ABB RAPID module: Module1_plano.mod

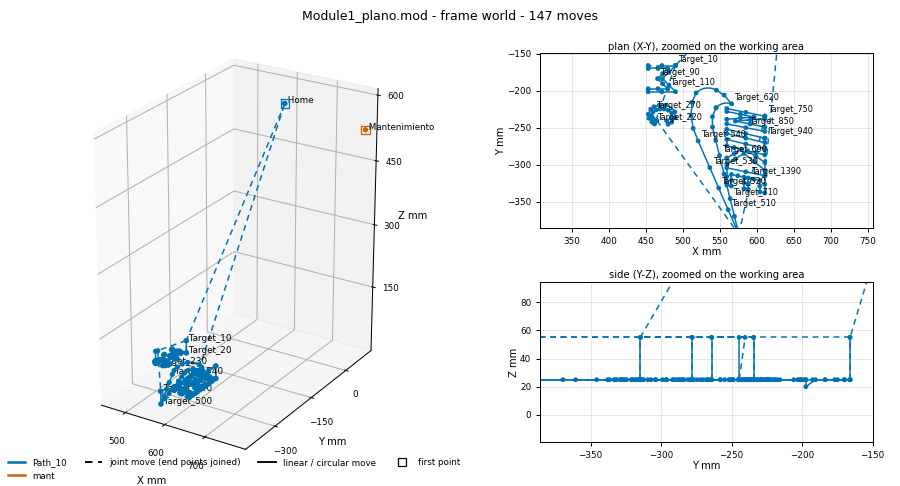
[picture p0: tool path of Module1_plano.mod in frame world, 147 of 147 moves have a stored position in this frame; points joined in program order, loops and branches not executed]
MODULE Module1
    PERS tooldata TCPTool_Lab1:=[TRUE,[[11.969,-5.577,162.232],[0.965925826,0,0.258819045,0]],[1,[0,0,1],[1,0,0,0],0,0,0]];
    TASK PERS wobjdata Workobject_2:=[FALSE,TRUE,"",[[667.5,-435,25],[0,0,1,0]],[[0,0,0],[1,0,0,0]]];
    CONST robtarget Target_10:=[[177.41,269.019,-30],[1,0,0,0],[0,0,-1,1],[9E+09,9E+09,9E+09,9E+09,9E+09,9E+09]];
    CONST robtarget Target_20:=[[177.41,269.019,0],[1,0,0,0],[0,0,-1,1],[9E+09,9E+09,9E+09,9E+09,9E+09,9E+09]];
    CONST robtarget Target_30:=[[195.844,269.019,0],[1,0,0,0],[0,0,-1,1],[9E+09,9E+09,9E+09,9E+09,9E+09,9E+09]];
    CONST robtarget Target_40:=[[214.279,269.019,0],[1,0,0,0],[0,0,-1,1],[9E+09,9E+09,9E+09,9E+09,9E+09,9E+09]];
    CONST robtarget Target_50:=[[214.279,265.019,0],[1,0,0,0],[0,0,-1,1],[9E+09,9E+09,9E+09,9E+09,9E+09,9E+09]];
    CONST robtarget Target_60:=[[201.112,265.019,0],[1,0,0,0],[0,0,-1,1],[9E+09,9E+09,9E+09,9E+09,9E+09,9E+09]];
    CONST robtarget Target_70:=[[187.944,265.019,0],[1,0,0,0],[0,0,-1,1],[9E+09,9E+09,9E+09,9E+09,9E+09,9E+09]];
    CONST robtarget Target_80:=[[194.783,258.18,0],[1,0,0,0],[0,0,-1,1],[9E+09,9E+09,9E+09,9E+09,9E+09,9E+09]];
    CONST robtarget Target_90:=[[201.622,251.341,0],[1,0,0,0],[0,0,-1,1],[9E+09,9E+09,9E+09,9E+09,9E+09,9E+09]];
    CONST robtarget Target_100:=[[194.783,244.503,0],[1,0,0,0],[0,0,-1,1],[9E+09,9E+09,9E+09,9E+09,9E+09,9E+09]];
    CONST robtarget Target_110:=[[187.944,237.664,5],[1,0,0,0],[0,0,-1,1],[9E+09,9E+09,9E+09,9E+09,9E+09,9E+09]];
    CONST robtarget Target_120:=[[201.112,237.664,0],[1,0,0,0],[0,0,-1,1],[9E+09,9E+09,9E+09,9E+09,9E+09,9E+09]];
    CONST robtarget Target_130:=[[214.279,237.664,0],[1,0,0,0],[0,0,-1,1],[9E+09,9E+09,9E+09,9E+09,9E+09,9E+09]];
    CONST robtarget Target_140:=[[214.279,233.664,0],[1,0,0,0],[0,0,-1,1],[9E+09,9E+09,9E+09,9E+09,9E+09,9E+09]];
    CONST robtarget Target_150:=[[195.844,233.664,0],[1,0,0,0],[0,0,-1,1],[9E+09,9E+09,9E+09,9E+09,9E+09,9E+09]];
    CONST robtarget Target_160:=[[177.41,233.664,0],[1,0,0,0],[0,0,-1,1],[9E+09,9E+09,9E+09,9E+09,9E+09,9E+09]];
    CONST robtarget Target_170:=[[186.248,242.503,0],[1,0,0,0],[0,0,-1,1],[9E+09,9E+09,9E+09,9E+09,9E+09,9E+09]];
    CONST robtarget Target_180:=[[195.087,251.341,0],[1,0,0,0],[0,0,-1,1],[9E+09,9E+09,9E+09,9E+09,9E+09,9E+09]];
    CONST robtarget Target_190:=[[186.248,260.18,0],[1,0,0,0],[0,0,-1,1],[9E+09,9E+09,9E+09,9E+09,9E+09,9E+09]];
    CONST robtarget Target_200:=[[177.41,269.019,0],[1,0,0,0],[0,0,-1,1],[9E+09,9E+09,9E+09,9E+09,9E+09,9E+09]];
    CONST robtarget Target_210:=[[177.41,269.019,-30],[1,0,0,0],[0,0,-1,1],[9E+09,9E+09,9E+09,9E+09,9E+09,9E+09]];
    CONST robtarget Target_220:=[[205.678,190.302,-30],[1,0,0,0],[0,0,-1,1],[9E+09,9E+09,9E+09,9E+09,9E+09,9E+09]];
    CONST robtarget Target_230:=[[205.623,190.276,0],[1,0,0,0],[0,0,-1,1],[9E+09,9E+09,9E+09,9E+09,9E+09,9E+09]];
    CONST robtarget Target_240:=[[202.955,194.702,0],[1,0,0,0],[0,0,-1,1],[9E+09,9E+09,9E+09,9E+09,9E+09,9E+09]];
    CONST robtarget Target_250:=[[207.34,197.113,0],[1,0,0,0],[0,0,-1,1],[9E+09,9E+09,9E+09,9E+09,9E+09,9E+09]];
    CONST robtarget Target_260:=[[209.847,201.03,0],[1,0,0,0],[0,0,-1,1],[9E+09,9E+09,9E+09,9E+09,9E+09,9E+09]];
    CONST robtarget Target_270:=[[208.011,206.295,0],[1,0,0,0],[0,0,-1,1],[9E+09,9E+09,9E+09,9E+09,9E+09,9E+09]];
    CONST robtarget Target_280:=[[203.511,209.124,0],[1,0,0,0],[0,0,-1,1],[9E+09,9E+09,9E+09,9E+09,9E+09,9E+09]];
    CONST robtarget Target_290:=[[198.638,210.318,0],[1,0,0,0],[0,0,-1,1],[9E+09,9E+09,9E+09,9E+09,9E+09,9E+09]];
    CONST robtarget Target_300:=[[192.941,210.304,0],[1,0,0,0],[0,0,-1,1],[9E+09,9E+09,9E+09,9E+09,9E+09,9E+09]];
    CONST robtarget Target_310:=[[187.344,208.773,0],[1,0,0,0],[0,0,-1,1],[9E+09,9E+09,9E+09,9E+09,9E+09,9E+09]];
    CONST robtarget Target_320:=[[182.65,205,0],[1,0,0,0],[0,0,-1,1],[9E+09,9E+09,9E+09,9E+09,9E+09,9E+09]];
    CONST robtarget Target_330:=[[182.874,198.696,0],[1,0,0,0],[0,0,-1,1],[9E+09,9E+09,9E+09,9E+09,9E+09,9E+09]];
    CONST robtarget Target_340:=[[189.379,194.489,0],[1,0,0,0],[0,0,-1,1],[9E+09,9E+09,9E+09,9E+09,9E+09,9E+09]];
    CONST robtarget Target_350:=[[187.41,189.702,0],[1,0,0,0],[0,0,-1,1],[9E+09,9E+09,9E+09,9E+09,9E+09,9E+09]];
    CONST robtarget Target_360:=[[182.414,192.529,0],[1,0,0,0],[0,0,-1,1],[9E+09,9E+09,9E+09,9E+09,9E+09,9E+09]];
    CONST robtarget Target_370:=[[178.043,198.417,0],[1,0,0,0],[0,0,-1,1],[9E+09,9E+09,9E+09,9E+09,9E+09,9E+09]];
    CONST robtarget Target_380:=[[178.344,206.368,0],[1,0,0,0],[0,0,-1,1],[9E+09,9E+09,9E+09,9E+09,9E+09,9E+09]];
    CONST robtarget Target_390:=[[182.556,211.614,0],[1,0,0,0],[0,0,-1,1],[9E+09,9E+09,9E+09,9E+09,9E+09,9E+09]];
    CONST robtarget Target_400:=[[190.831,215.342,0],[1,0,0,0],[0,0,-1,1],[9E+09,9E+09,9E+09,9E+09,9E+09,9E+09]];
    CONST robtarget Target_410:=[[199.222,215.629,0],[1,0,0,0],[0,0,-1,1],[9E+09,9E+09,9E+09,9E+09,9E+09,9E+09]];
    CONST robtarget Target_420:=[[206.382,213.378,0],[1,0,0,0],[0,0,-1,1],[9E+09,9E+09,9E+09,9E+09,9E+09,9E+09]];
    CONST robtarget Target_430:=[[210.902,210.005,0],[1,0,0,0],[0,0,-1,1],[9E+09,9E+09,9E+09,9E+09,9E+09,9E+09]];
    CONST robtarget Target_440:=[[214.199,203.307,0],[1,0,0,0],[0,0,-1,1],[9E+09,9E+09,9E+09,9E+09,9E+09,9E+09]];
    CONST robtarget Target_450:=[[213.42,197.838,0],[1,0,0,0],[0,0,-1,1],[9E+09,9E+09,9E+09,9E+09,9E+09,9E+09]];
    CONST robtarget Target_460:=[[209.362,192.6,0],[1,0,0,0],[0,0,-1,1],[9E+09,9E+09,9E+09,9E+09,9E+09,9E+09]];
    CONST robtarget Target_470:=[[205.915,190.416,0],[1,0,0,0],[0,0,-1,1],[9E+09,9E+09,9E+09,9E+09,9E+09,9E+09]];
    CONST robtarget Target_480:=[[202.627,194.59,-30],[1,0,0,0],[0,0,-1,1],[9E+09,9E+09,9E+09,9E+09,9E+09,9E+09]];
    CONST robtarget Target_490:=[[91.883,41.213,-30],[1,0,0,0],[-1,-1,0,1],[9E+09,9E+09,9E+09,9E+09,9E+09,9E+09]];
    CONST robtarget Target_500:=[[91.883,41.213,0],[1,0,0,0],[-1,-1,0,1],[9E+09,9E+09,9E+09,9E+09,9E+09,9E+09]];
    CONST robtarget Target_510:=[[106.332,74.333,0],[1,0,0,0],[-1,-1,0,1],[9E+09,9E+09,9E+09,9E+09,9E+09,9E+09]];
    CONST robtarget Target_520:=[[119.103,103.607,0],[1,0,0,0],[-1,-1,0,1],[9E+09,9E+09,9E+09,9E+09,9E+09,9E+09]];
    CONST robtarget Target_530:=[[131.177,131.283,0],[1,0,0,0],[0,0,-1,1],[9E+09,9E+09,9E+09,9E+09,9E+09,9E+09]];
    CONST robtarget Target_540:=[[146.843,167.193,0],[1,0,0,0],[0,0,-1,1],[9E+09,9E+09,9E+09,9E+09,9E+09,9E+09]];
    CONST robtarget Target_550:=[[153.569,184.183,0],[1,0,0,0],[0,0,-1,1],[9E+09,9E+09,9E+09,9E+09,9E+09,9E+09]];
    CONST robtarget Target_560:=[[156.337,201.217,0],[1,0,0,0],[0,0,-1,1],[9E+09,9E+09,9E+09,9E+09,9E+09,9E+09]];
    CONST robtarget Target_570:=[[155.288,219.26,0],[1,0,0,0],[0,0,-1,1],[9E+09,9E+09,9E+09,9E+09,9E+09,9E+09]];
    CONST robtarget Target_580:=[[149.597,231.965,0],[1,0,0,0],[0,0,-1,1],[9E+09,9E+09,9E+09,9E+09,9E+09,9E+09]];
    CONST robtarget Target_590:=[[140.915,237.42,0],[1,0,0,0],[0,0,-1,1],[9E+09,9E+09,9E+09,9E+09,9E+09,9E+09]];
    CONST robtarget Target_600:=[[122.252,235.701,0],[1,0,0,0],[0,0,-1,1],[9E+09,9E+09,9E+09,9E+09,9E+09,9E+09]];
    CONST robtarget Target_610:=[[111.771,229.081,0],[1,0,0,0],[0,0,-1,1],[9E+09,9E+09,9E+09,9E+09,9E+09,9E+09]];
    CONST robtarget Target_620:=[[101.618,217.264,0],[1,0,0,0],[0,0,-1,1],[9E+09,9E+09,9E+09,9E+09,9E+09,9E+09]];
    CONST robtarget Target_630:=[[112.39,217.915,0],[1,0,0,0],[0,0,-1,1],[9E+09,9E+09,9E+09,9E+09,9E+09,9E+09]];
    CONST robtarget Target_640:=[[122.65,212.032,0],[1,0,0,0],[0,0,-1,1],[9E+09,9E+09,9E+09,9E+09,9E+09,9E+09]];
    CONST robtarget Target_650:=[[122.562,212.129,0],[1,0,0,0],[0,0,-1,1],[9E+09,9E+09,9E+09,9E+09,9E+09,9E+09]];
    CONST robtarget Target_660:=[[127.578,199.979,0],[1,0,0,0],[0,0,-1,1],[9E+09,9E+09,9E+09,9E+09,9E+09,9E+09]];
    CONST robtarget Target_670:=[[127.52,186.008,0],[1,0,0,0],[0,0,-1,1],[9E+09,9E+09,9E+09,9E+09,9E+09,9E+09]];
    CONST robtarget Target_680:=[[123.036,167.787,0],[1,0,0,0],[0,0,-1,1],[9E+09,9E+09,9E+09,9E+09,9E+09,9E+09]];
    CONST robtarget Target_690:=[[118.036,147.473,0],[1,0,0,0],[0,0,-1,1],[9E+09,9E+09,9E+09,9E+09,9E+09,9E+09]];
    CONST robtarget Target_700:=[[111.892,122.51,0],[1,0,0,0],[-1,-1,0,1],[9E+09,9E+09,9E+09,9E+09,9E+09,9E+09]];
    CONST robtarget Target_710:=[[103.706,89.25,0],[1,0,0,0],[-1,-1,0,1],[9E+09,9E+09,9E+09,9E+09,9E+09,9E+09]];
    CONST robtarget Target_720:=[[97.833,65.387,0],[1,0,0,0],[-1,-1,0,1],[9E+09,9E+09,9E+09,9E+09,9E+09,9E+09]];
    CONST robtarget Target_730:=[[91.883,41.213,0],[1,0,0,0],[-1,-1,0,1],[9E+09,9E+09,9E+09,9E+09,9E+09,9E+09]];
    CONST robtarget Target_740:=[[91.883,41.213,-30],[1,0,0,0],[-1,-1,0,1],[9E+09,9E+09,9E+09,9E+09,9E+09,9E+09]];
    CONST robtarget Target_750:=[[56.869,200.624,-30],[1,0,0,0],[0,0,-1,1],[9E+09,9E+09,9E+09,9E+09,9E+09,9E+09]];
    CONST robtarget Target_760:=[[56.869,200.624,0],[1,0,0,0],[0,0,-1,1],[9E+09,9E+09,9E+09,9E+09,9E+09,9E+09]];
    CONST robtarget Target_770:=[[82.551,205.76,0],[1,0,0,0],[0,0,-1,1],[9E+09,9E+09,9E+09,9E+09,9E+09,9E+09]];
    CONST robtarget Target_780:=[[108.233,210.896,0],[1,0,0,0],[0,0,-1,1],[9E+09,9E+09,9E+09,9E+09,9E+09,9E+09]];
    CONST robtarget Target_790:=[[108.233,206.964,0],[1,0,0,0],[0,0,-1,1],[9E+09,9E+09,9E+09,9E+09,9E+09,9E+09]];
    CONST robtarget Target_800:=[[89.785,203.274,0],[1,0,0,0],[0,0,-1,1],[9E+09,9E+09,9E+09,9E+09,9E+09,9E+09]];
    CONST robtarget Target_810:=[[71.337,199.585,0],[1,0,0,0],[0,0,-1,1],[9E+09,9E+09,9E+09,9E+09,9E+09,9E+09]];
    CONST robtarget Target_820:=[[89.785,198.008,0],[1,0,0,0],[0,0,-1,1],[9E+09,9E+09,9E+09,9E+09,9E+09,9E+09]];
    CONST robtarget Target_830:=[[108.233,196.431,0],[1,0,0,0],[0,0,-1,1],[9E+09,9E+09,9E+09,9E+09,9E+09,9E+09]];
    CONST robtarget Target_840:=[[108.233,190.27,0],[1,0,0,0],[0,0,-1,1],[9E+09,9E+09,9E+09,9E+09,9E+09,9E+09]];
    CONST robtarget Target_850:=[[82.554,185.135,0],[1,0,0,0],[0,0,-1,1],[9E+09,9E+09,9E+09,9E+09,9E+09,9E+09]];
    CONST robtarget Target_860:=[[56.875,179.999,0],[1,0,0,0],[0,0,-1,1],[9E+09,9E+09,9E+09,9E+09,9E+09,9E+09]];
    CONST robtarget Target_870:=[[56.875,186.086,0],[1,0,0,0],[0,0,-1,1],[9E+09,9E+09,9E+09,9E+09,9E+09,9E+09]];
    CONST robtarget Target_880:=[[76.742,190.059,0],[1,0,0,0],[0,0,-1,1],[9E+09,9E+09,9E+09,9E+09,9E+09,9E+09]];
    CONST robtarget Target_890:=[[96.61,194.033,0],[1,0,0,0],[0,0,-1,1],[9E+09,9E+09,9E+09,9E+09,9E+09,9E+09]];
    CONST robtarget Target_900:=[[76.742,195.731,0],[1,0,0,0],[0,0,-1,1],[9E+09,9E+09,9E+09,9E+09,9E+09,9E+09]];
    CONST robtarget Target_910:=[[56.875,197.429,0],[1,0,0,0],[0,0,-1,1],[9E+09,9E+09,9E+09,9E+09,9E+09,9E+09]];
    CONST robtarget Target_920:=[[56.869,200.624,0],[1,0,0,0],[0,0,-1,1],[9E+09,9E+09,9E+09,9E+09,9E+09,9E+09]];
    CONST robtarget Target_930:=[[56.869,200.624,-30],[1,0,0,0],[0,0,-1,1],[9E+09,9E+09,9E+09,9E+09,9E+09,9E+09]];
    CONST robtarget Target_940:=[[56.875,170.875,-30],[1,0,0,0],[0,0,-1,1],[9E+09,9E+09,9E+09,9E+09,9E+09,9E+09]];
    CONST robtarget Target_950:=[[56.875,170.875,0],[1,0,0,0],[0,0,-1,1],[9E+09,9E+09,9E+09,9E+09,9E+09,9E+09]];
    CONST robtarget Target_960:=[[82.554,176.959,0],[1,0,0,0],[0,0,-1,1],[9E+09,9E+09,9E+09,9E+09,9E+09,9E+09]];
    CONST robtarget Target_970:=[[108.233,183.043,0],[1,0,0,0],[0,0,-1,1],[9E+09,9E+09,9E+09,9E+09,9E+09,9E+09]];
    CONST robtarget Target_980:=[[108.233,177.043,0],[1,0,0,0],[0,0,-1,1],[9E+09,9E+09,9E+09,9E+09,9E+09,9E+09]];
    CONST robtarget Target_990:=[[82.554,170.959,0],[1,0,0,0],[0,0,-1,1],[9E+09,9E+09,9E+09,9E+09,9E+09,9E+09]];
    CONST robtarget Target_1000:=[[56.875,164.875,0],[1,0,0,0],[0,0,-1,1],[9E+09,9E+09,9E+09,9E+09,9E+09,9E+09]];
    CONST robtarget Target_1010:=[[56.875,170.875,0],[1,0,0,0],[0,0,-1,1],[9E+09,9E+09,9E+09,9E+09,9E+09,9E+09]];
    CONST robtarget Target_1020:=[[56.875,170.875,-30],[1,0,0,0],[0,0,-1,1],[9E+09,9E+09,9E+09,9E+09,9E+09,9E+09]];
    CONST robtarget Target_1030:=[[56.875,157.002,-30],[1,0,0,0],[0,0,-1,1],[9E+09,9E+09,9E+09,9E+09,9E+09,9E+09]];
    CONST robtarget Target_1040:=[[56.875,157.002,0],[1,0,0,0],[0,0,-1,1],[9E+09,9E+09,9E+09,9E+09,9E+09,9E+09]];
    CONST robtarget Target_1050:=[[82.554,163.085,0],[1,0,0,0],[0,0,-1,1],[9E+09,9E+09,9E+09,9E+09,9E+09,9E+09]];
    CONST robtarget Target_1060:=[[108.233,169.169,0],[1,0,0,0],[0,0,-1,1],[9E+09,9E+09,9E+09,9E+09,9E+09,9E+09]];
    CONST robtarget Target_1070:=[[108.233,160.652,0],[1,0,0,0],[0,0,-1,1],[9E+09,9E+09,9E+09,9E+09,9E+09,9E+09]];
    CONST robtarget Target_1080:=[[98.214,158.278,0],[1,0,0,0],[0,0,-1,1],[9E+09,9E+09,9E+09,9E+09,9E+09,9E+09]];
    CONST robtarget Target_1090:=[[88.195,155.905,0],[1,0,0,0],[0,0,-1,1],[9E+09,9E+09,9E+09,9E+09,9E+09,9E+09]];
    CONST robtarget Target_1100:=[[98.214,150.082,0],[1,0,0,0],[0,0,-1,1],[9E+09,9E+09,9E+09,9E+09,9E+09,9E+09]];
    CONST robtarget Target_1110:=[[108.233,144.259,0],[1,0,0,0],[0,0,-1,1],[9E+09,9E+09,9E+09,9E+09,9E+09,9E+09]];
    CONST robtarget Target_1120:=[[108.233,135.914,0],[1,0,0,0],[0,0,-1,1],[9E+09,9E+09,9E+09,9E+09,9E+09,9E+09]];
    CONST robtarget Target_1130:=[[96.587,143.111,0],[1,0,0,0],[0,0,-1,1],[9E+09,9E+09,9E+09,9E+09,9E+09,9E+09]];
    CONST robtarget Target_1140:=[[84.942,150.308,0],[1,0,0,0],[0,0,-1,1],[9E+09,9E+09,9E+09,9E+09,9E+09,9E+09]];
    CONST robtarget Target_1150:=[[70.909,139.04,0],[1,0,0,0],[0,0,-1,1],[9E+09,9E+09,9E+09,9E+09,9E+09,9E+09]];
    CONST robtarget Target_1160:=[[56.875,127.772,0],[1,0,0,0],[-1,-1,0,1],[9E+09,9E+09,9E+09,9E+09,9E+09,9E+09]];
    CONST robtarget Target_1170:=[[56.875,138.348,0],[1,0,0,0],[0,0,-1,1],[9E+09,9E+09,9E+09,9E+09,9E+09,9E+09]];
    CONST robtarget Target_1180:=[[68.658,146.208,0],[1,0,0,0],[0,0,-1,1],[9E+09,9E+09,9E+09,9E+09,9E+09,9E+09]];
    CONST robtarget Target_1190:=[[80.44,154.068,0],[1,0,0,0],[0,0,-1,1],[9E+09,9E+09,9E+09,9E+09,9E+09,9E+09]];
    CONST robtarget Target_1200:=[[68.658,151.276,0],[1,0,0,0],[0,0,-1,1],[9E+09,9E+09,9E+09,9E+09,9E+09,9E+09]];
    CONST robtarget Target_1210:=[[56.875,148.485,0],[1,0,0,0],[0,0,-1,1],[9E+09,9E+09,9E+09,9E+09,9E+09,9E+09]];
    CONST robtarget Target_1220:=[[56.875,157.002,0],[1,0,0,0],[0,0,-1,1],[9E+09,9E+09,9E+09,9E+09,9E+09,9E+09]];
    CONST robtarget Target_1230:=[[56.875,157.002,-30],[1,0,0,0],[0,0,-1,1],[9E+09,9E+09,9E+09,9E+09,9E+09,9E+09]];
    CONST robtarget Target_1240:=[[56.875,120.255,-30],[1,0,0,0],[-1,-1,0,1],[9E+09,9E+09,9E+09,9E+09,9E+09,9E+09]];
    CONST robtarget Target_1250:=[[56.875,120.255,0],[1,0,0,0],[-1,-1,0,1],[9E+09,9E+09,9E+09,9E+09,9E+09,9E+09]];
    CONST robtarget Target_1260:=[[82.554,125.558,0],[1,0,0,0],[-1,-1,0,1],[9E+09,9E+09,9E+09,9E+09,9E+09,9E+09]];
    CONST robtarget Target_1270:=[[108.233,130.861,0],[1,0,0,0],[0,0,-1,1],[9E+09,9E+09,9E+09,9E+09,9E+09,9E+09]];
    CONST robtarget Target_1280:=[[108.233,119.251,0],[1,0,0,0],[-1,-1,0,1],[9E+09,9E+09,9E+09,9E+09,9E+09,9E+09]];
    CONST robtarget Target_1290:=[[108.233,107.642,0],[1,0,0,0],[-1,-1,0,1],[9E+09,9E+09,9E+09,9E+09,9E+09,9E+09]];
    CONST robtarget Target_1300:=[[101.866,106.328,0],[1,0,0,0],[-1,-1,0,1],[9E+09,9E+09,9E+09,9E+09,9E+09,9E+09]];
    CONST robtarget Target_1310:=[[101.866,114.138,0],[1,0,0,0],[-1,-1,0,1],[9E+09,9E+09,9E+09,9E+09,9E+09,9E+09]];
    CONST robtarget Target_1320:=[[101.866,121.949,0],[1,0,0,0],[-1,-1,0,1],[9E+09,9E+09,9E+09,9E+09,9E+09,9E+09]];
    CONST robtarget Target_1330:=[[93.404,120.169,0],[1,0,0,0],[-1,-1,0,1],[9E+09,9E+09,9E+09,9E+09,9E+09,9E+09]];
    CONST robtarget Target_1340:=[[84.942,118.39,0],[1,0,0,0],[-1,-1,0,1],[9E+09,9E+09,9E+09,9E+09,9E+09,9E+09]];
    CONST robtarget Target_1350:=[[84.942,110.611,0],[1,0,0,0],[-1,-1,0,1],[9E+09,9E+09,9E+09,9E+09,9E+09,9E+09]];
    CONST robtarget Target_1360:=[[84.942,102.833,0],[1,0,0,0],[-1,-1,0,1],[9E+09,9E+09,9E+09,9E+09,9E+09,9E+09]];
    CONST robtarget Target_1370:=[[79.224,101.652,0],[1,0,0,0],[-1,-1,0,1],[9E+09,9E+09,9E+09,9E+09,9E+09,9E+09]];
    CONST robtarget Target_1380:=[[79.224,109.42,0],[1,0,0,0],[-1,-1,0,1],[9E+09,9E+09,9E+09,9E+09,9E+09,9E+09]];
    CONST robtarget Target_1390:=[[79.224,117.187,0],[1,0,0,0],[-1,-1,0,1],[9E+09,9E+09,9E+09,9E+09,9E+09,9E+09]];
    CONST robtarget Target_1400:=[[71.411,115.544,0],[1,0,0,0],[-1,-1,0,1],[9E+09,9E+09,9E+09,9E+09,9E+09,9E+09]];
    CONST robtarget Target_1410:=[[63.597,113.901,0],[1,0,0,0],[-1,-1,0,1],[9E+09,9E+09,9E+09,9E+09,9E+09,9E+09]];
    CONST robtarget Target_1420:=[[63.597,106.163,0],[1,0,0,0],[-1,-1,0,1],[9E+09,9E+09,9E+09,9E+09,9E+09,9E+09]];
    CONST robtarget Target_1430:=[[63.597,98.425,0],[1,0,0,0],[-1,-1,0,1],[9E+09,9E+09,9E+09,9E+09,9E+09,9E+09]];
    CONST robtarget Target_1440:=[[56.875,97.037,0],[1,0,0,0],[-1,-1,0,1],[9E+09,9E+09,9E+09,9E+09,9E+09,9E+09]];
    CONST robtarget Target_1450:=[[56.875,108.646,0],[1,0,0,0],[-1,-1,0,1],[9E+09,9E+09,9E+09,9E+09,9E+09,9E+09]];
    CONST robtarget Target_1460:=[[56.875,120.255,0],[1,0,0,0],[-1,-1,0,1],[9E+09,9E+09,9E+09,9E+09,9E+09,9E+09]];
    CONST robtarget Target_1470:=[[56.875,120.255,-30],[1,0,0,0],[-1,-1,0,1],[9E+09,9E+09,9E+09,9E+09,9E+09,9E+09]];
    CONST robtarget Home:=[[26.695815447,429.423,-563.018541942],[0.965925826,0,-0.258819045,0],[-1,0,-1,0],[9E+09,9E+09,9E+09,9E+09,9E+09,9E+09]];
    CONST robtarget Home_2:=[[74.783200826,129.426583542,-420.91739945],[0.993217397,0.000004228,0.116272108,0.000000495],[0,1,-2,1],[9E+09,9E+09,9E+09,9E+09,9E+09,9E+09]];
    CONST robtarget Mantenimiento:=[[-116.188,526.934,-500.556],[0.924164952,-0.278371196,-0.154994418,-0.210725769],[0,0,-1,0],[9E+09,9E+09,9E+09,9E+09,9E+09,9E+09]];
    CONST robtarget Home_1:=[[-77.086561778,129.419166281,-428.818733092],[0.993216571,-0.00000444,0.11627916,-0.00000052],[-1,0,-1,0],[9E+09,9E+09,9E+09,9E+09,9E+09,9E+09]];

    PROC Path_10()
        MoveJ Home,v200,z5,TCPTool_Lab1\WObj:=Workobject_2;
        MoveJ Target_10,v200,z5,TCPTool_Lab1\WObj:=Workobject_2;
        MoveL Target_20,v200,fine,TCPTool_Lab1\WObj:=Workobject_2;
        MoveL Target_30,v100,z0,TCPTool_Lab1\WObj:=Workobject_2;
        MoveJ Target_40,v100,z0,TCPTool_Lab1\WObj:=Workobject_2;
        MoveL Target_50,v100,z0,TCPTool_Lab1\WObj:=Workobject_2;
        MoveL Target_60,v100,z0,TCPTool_Lab1\WObj:=Workobject_2;
        MoveL Target_70,v100,z0,TCPTool_Lab1\WObj:=Workobject_2;
        MoveL Target_80,v100,z0,TCPTool_Lab1\WObj:=Workobject_2;
        MoveL Target_90,v100,z0,TCPTool_Lab1\WObj:=Workobject_2;
        MoveL Target_100,v100,z0,TCPTool_Lab1\WObj:=Workobject_2;
        MoveL Target_110,v100,z0,TCPTool_Lab1\WObj:=Workobject_2;
        MoveL Target_120,v100,z0,TCPTool_Lab1\WObj:=Workobject_2;
        MoveL Target_130,v100,z0,TCPTool_Lab1\WObj:=Workobject_2;
        MoveL Target_140,v100,z0,TCPTool_Lab1\WObj:=Workobject_2;
        MoveL Target_150,v100,z0,TCPTool_Lab1\WObj:=Workobject_2;
        MoveL Target_160,v100,z0,TCPTool_Lab1\WObj:=Workobject_2;
        MoveL Target_170,v100,z0,TCPTool_Lab1\WObj:=Workobject_2;
        MoveL Target_180,v100,z0,TCPTool_Lab1\WObj:=Workobject_2;
        MoveL Target_190,v100,z0,TCPTool_Lab1\WObj:=Workobject_2;
        MoveL Target_200,v100,z0,TCPTool_Lab1\WObj:=Workobject_2;
        MoveJ Target_210,v200,z5,TCPTool_Lab1\WObj:=Workobject_2;
        MoveJ Target_220,v200,z5,TCPTool_Lab1\WObj:=Workobject_2;
        MoveL Target_230,v100,fine,TCPTool_Lab1\WObj:=Workobject_2;
        MoveL Target_240,v100,z0,TCPTool_Lab1\WObj:=Workobject_2;
        MoveL Target_250,v100,z0,TCPTool_Lab1\WObj:=Workobject_2;
        MoveL Target_260,v100,z0,TCPTool_Lab1\WObj:=Workobject_2;
        MoveL Target_270,v100,z0,TCPTool_Lab1\WObj:=Workobject_2;
        MoveL Target_280,v100,z0,TCPTool_Lab1\WObj:=Workobject_2;
        MoveL Target_290,v100,z0,TCPTool_Lab1\WObj:=Workobject_2;
        MoveL Target_300,v100,z0,TCPTool_Lab1\WObj:=Workobject_2;
        MoveL Target_310,v100,z0,TCPTool_Lab1\WObj:=Workobject_2;
        MoveL Target_320,v100,z0,TCPTool_Lab1\WObj:=Workobject_2;
        MoveL Target_330,v100,z0,TCPTool_Lab1\WObj:=Workobject_2;
        MoveL Target_340,v100,z0,TCPTool_Lab1\WObj:=Workobject_2;
        MoveL Target_350,v100,z0,TCPTool_Lab1\WObj:=Workobject_2;
        MoveL Target_360,v100,z0,TCPTool_Lab1\WObj:=Workobject_2;
        MoveL Target_370,v100,z0,TCPTool_Lab1\WObj:=Workobject_2;
        MoveL Target_380,v100,z0,TCPTool_Lab1\WObj:=Workobject_2;
        MoveC Target_390,Target_400,v100,z0,TCPTool_Lab1\WObj:=Workobject_2;
        MoveL Target_410,v100,z0,TCPTool_Lab1\WObj:=Workobject_2;
        MoveL Target_420,v100,z0,TCPTool_Lab1\WObj:=Workobject_2;
        MoveL Target_430,v100,z0,TCPTool_Lab1\WObj:=Workobject_2;
        MoveL Target_440,v100,z0,TCPTool_Lab1\WObj:=Workobject_2;
        MoveL Target_450,v100,z0,TCPTool_Lab1\WObj:=Workobject_2;
        MoveL Target_460,v100,z0,TCPTool_Lab1\WObj:=Workobject_2;
        MoveL Target_470,v100,z0,TCPTool_Lab1\WObj:=Workobject_2;
        MoveJ Target_480,v200,z5,TCPTool_Lab1\WObj:=Workobject_2;
        MoveJ Target_490,v200,z5,TCPTool_Lab1\WObj:=Workobject_2;
        MoveL Target_500,v100,fine,TCPTool_Lab1\WObj:=Workobject_2;
        MoveL Target_510,v100,z0,TCPTool_Lab1\WObj:=Workobject_2;
        MoveL Target_520,v100,z0,TCPTool_Lab1\WObj:=Workobject_2;
        MoveL Target_530,v100,z0,TCPTool_Lab1\WObj:=Workobject_2;
        MoveL Target_540,v100,z0,TCPTool_Lab1\WObj:=Workobject_2;
        MoveL Target_550,v100,z0,TCPTool_Lab1\WObj:=Workobject_2;
        MoveL Target_560,v100,z0,TCPTool_Lab1\WObj:=Workobject_2;
        MoveL Target_570,v100,z0,TCPTool_Lab1\WObj:=Workobject_2;
        MoveL Target_580,v100,z0,TCPTool_Lab1\WObj:=Workobject_2;
        MoveC Target_590,Target_600,v100,z0,TCPTool_Lab1\WObj:=Workobject_2;
        MoveL Target_610,v100,z0,TCPTool_Lab1\WObj:=Workobject_2;
        MoveL Target_620,v100,z0,TCPTool_Lab1\WObj:=Workobject_2;
        MoveC Target_630,Target_640,v100,z0,TCPTool_Lab1\WObj:=Workobject_2;
        MoveL Target_650,v100,z0,TCPTool_Lab1\WObj:=Workobject_2;
        MoveL Target_660,v100,z0,TCPTool_Lab1\WObj:=Workobject_2;
        MoveL Target_670,v100,z0,TCPTool_Lab1\WObj:=Workobject_2;
        MoveL Target_680,v100,z0,TCPTool_Lab1\WObj:=Workobject_2;
        MoveL Target_690,v100,z0,TCPTool_Lab1\WObj:=Workobject_2;
        MoveL Target_700,v100,z0,TCPTool_Lab1\WObj:=Workobject_2;
        MoveL Target_710,v100,z0,TCPTool_Lab1\WObj:=Workobject_2;
        MoveL Target_720,v100,z0,TCPTool_Lab1\WObj:=Workobject_2;
        MoveL Target_730,v100,z0,TCPTool_Lab1\WObj:=Workobject_2;
        MoveJ Target_740,v200,z5,TCPTool_Lab1\WObj:=Workobject_2;
        MoveJ Target_750,v200,z5,TCPTool_Lab1\WObj:=Workobject_2;
        MoveL Target_760,v100,fine,TCPTool_Lab1\WObj:=Workobject_2;
        MoveL Target_770,v100,z0,TCPTool_Lab1\WObj:=Workobject_2;
        MoveL Target_780,v100,z0,TCPTool_Lab1\WObj:=Workobject_2;
        MoveL Target_790,v100,z0,TCPTool_Lab1\WObj:=Workobject_2;
        MoveL Target_800,v100,z0,TCPTool_Lab1\WObj:=Workobject_2;
        MoveL Target_810,v100,z0,TCPTool_Lab1\WObj:=Workobject_2;
        MoveL Target_820,v100,z0,TCPTool_Lab1\WObj:=Workobject_2;
        MoveL Target_830,v100,z0,TCPTool_Lab1\WObj:=Workobject_2;
        MoveL Target_840,v100,z0,TCPTool_Lab1\WObj:=Workobject_2;
        MoveL Target_850,v100,z0,TCPTool_Lab1\WObj:=Workobject_2;
        MoveL Target_860,v100,z0,TCPTool_Lab1\WObj:=Workobject_2;
        MoveL Target_870,v100,z0,TCPTool_Lab1\WObj:=Workobject_2;
        MoveL Target_880,v100,z0,TCPTool_Lab1\WObj:=Workobject_2;
        MoveL Target_890,v100,z0,TCPTool_Lab1\WObj:=Workobject_2;
        MoveL Target_900,v100,z0,TCPTool_Lab1\WObj:=Workobject_2;
        MoveL Target_910,v100,z0,TCPTool_Lab1\WObj:=Workobject_2;
        MoveL Target_920,v100,z0,TCPTool_Lab1\WObj:=Workobject_2;
        MoveJ Target_930,v200,z5,TCPTool_Lab1\WObj:=Workobject_2;
        MoveJ Target_940,v200,z5,TCPTool_Lab1\WObj:=Workobject_2;
        MoveL Target_950,v100,fine,TCPTool_Lab1\WObj:=Workobject_2;
        MoveL Target_960,v100,z0,TCPTool_Lab1\WObj:=Workobject_2;
        MoveL Target_970,v100,z0,TCPTool_Lab1\WObj:=Workobject_2;
        MoveL Target_980,v100,z0,TCPTool_Lab1\WObj:=Workobject_2;
        MoveL Target_990,v100,z0,TCPTool_Lab1\WObj:=Workobject_2;
        MoveL Target_1000,v100,z0,TCPTool_Lab1\WObj:=Workobject_2;
        MoveL Target_1010,v100,z0,TCPTool_Lab1\WObj:=Workobject_2;
        MoveJ Target_1020,v200,z5,TCPTool_Lab1\WObj:=Workobject_2;
        MoveJ Target_1030,v200,z5,TCPTool_Lab1\WObj:=Workobject_2;
        MoveL Target_1040,v100,fine,TCPTool_Lab1\WObj:=Workobject_2;
        MoveL Target_1050,v100,z0,TCPTool_Lab1\WObj:=Workobject_2;
        MoveL Target_1060,v100,z0,TCPTool_Lab1\WObj:=Workobject_2;
        MoveL Target_1070,v100,z0,TCPTool_Lab1\WObj:=Workobject_2;
        MoveL Target_1080,v100,z0,TCPTool_Lab1\WObj:=Workobject_2;
        MoveL Target_1090,v100,z0,TCPTool_Lab1\WObj:=Workobject_2;
        MoveL Target_1100,v100,z0,TCPTool_Lab1\WObj:=Workobject_2;
        MoveL Target_1110,v100,z0,TCPTool_Lab1\WObj:=Workobject_2;
        MoveL Target_1120,v100,z0,TCPTool_Lab1\WObj:=Workobject_2;
        MoveL Target_1130,v100,z0,TCPTool_Lab1\WObj:=Workobject_2;
        MoveL Target_1140,v100,z0,TCPTool_Lab1\WObj:=Workobject_2;
        MoveL Target_1150,v100,z0,TCPTool_Lab1\WObj:=Workobject_2;
        MoveL Target_1160,v100,z0,TCPTool_Lab1\WObj:=Workobject_2;
        MoveL Target_1170,v100,z0,TCPTool_Lab1\WObj:=Workobject_2;
        MoveL Target_1180,v100,z0,TCPTool_Lab1\WObj:=Workobject_2;
        MoveL Target_1190,v100,z0,TCPTool_Lab1\WObj:=Workobject_2;
        MoveL Target_1200,v100,z0,TCPTool_Lab1\WObj:=Workobject_2;
        MoveL Target_1210,v100,z0,TCPTool_Lab1\WObj:=Workobject_2;
        MoveL Target_1220,v100,z0,TCPTool_Lab1\WObj:=Workobject_2;
        MoveJ Target_1230,v200,z5,TCPTool_Lab1\WObj:=Workobject_2;
        MoveJ Target_1240,v200,z5,TCPTool_Lab1\WObj:=Workobject_2;
        MoveL Target_1250,v100,fine,TCPTool_Lab1\WObj:=Workobject_2;
        MoveL Target_1260,v100,z0,TCPTool_Lab1\WObj:=Workobject_2;
        MoveL Target_1270,v100,z0,TCPTool_Lab1\WObj:=Workobject_2;
        MoveL Target_1280,v100,z0,TCPTool_Lab1\WObj:=Workobject_2;
        MoveL Target_1290,v100,z0,TCPTool_Lab1\WObj:=Workobject_2;
        MoveL Target_1300,v100,z0,TCPTool_Lab1\WObj:=Workobject_2;
        MoveL Target_1310,v100,z0,TCPTool_Lab1\WObj:=Workobject_2;
        MoveL Target_1320,v100,z0,TCPTool_Lab1\WObj:=Workobject_2;
        MoveL Target_1330,v100,z0,TCPTool_Lab1\WObj:=Workobject_2;
        MoveL Target_1340,v100,z0,TCPTool_Lab1\WObj:=Workobject_2;
        MoveL Target_1350,v100,z0,TCPTool_Lab1\WObj:=Workobject_2;
        MoveL Target_1360,v100,z0,TCPTool_Lab1\WObj:=Workobject_2;
        MoveL Target_1370,v100,z0,TCPTool_Lab1\WObj:=Workobject_2;
        MoveL Target_1380,v100,z0,TCPTool_Lab1\WObj:=Workobject_2;
        MoveL Target_1390,v100,z0,TCPTool_Lab1\WObj:=Workobject_2;
        MoveL Target_1400,v100,z0,TCPTool_Lab1\WObj:=Workobject_2;
        MoveL Target_1410,v100,z0,TCPTool_Lab1\WObj:=Workobject_2;
        MoveL Target_1420,v100,z0,TCPTool_Lab1\WObj:=Workobject_2;
        MoveL Target_1430,v100,z0,TCPTool_Lab1\WObj:=Workobject_2;
        MoveL Target_1440,v100,z0,TCPTool_Lab1\WObj:=Workobject_2;
        MoveL Target_1450,v100,z0,TCPTool_Lab1\WObj:=Workobject_2;
        MoveL Target_1460,v100,z0,TCPTool_Lab1\WObj:=Workobject_2;
        MoveJ Target_1470,v200,z5,TCPTool_Lab1\WObj:=Workobject_2;
        MoveJ Home,v200,z5,TCPTool_Lab1\WObj:=Workobject_2;
    ENDPROC

    PROC mant()
        MoveJ Mantenimiento,v200,z5,TCPTool_Lab1\WObj:=Workobject_2;
    ENDPROC

    PROC main()
    WHILE TRUE DO
        IF DI_01=1 THEN
            SetDO DO_01,1;
            SetDO DO_01,0;
            Path_10;
            STOP;
        ELSE IF DI_02=1 THEN
            SetDO DO_01,0;
            SetDO DO_01,1;
            mant;
            STOP;
        ENDIF
      ENDIF
    ENDWHILE
ENDPROC
ENDMODULE
